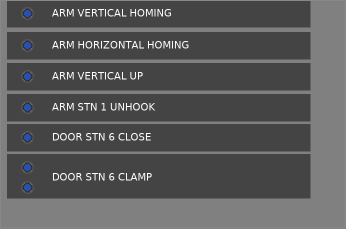
VISUALIZATION Popup_OriginStatus  // 346x229
    Rectangle (0,0 346x229)
    Rectangle (7,0 303x27)
    Label (49,1 258x24), "ARM VERTICAL HOMING"
    Lamp1 (20,6 15x15), variable: ARbArmVertHomeDone[1], style: Lamp-Lamp1-Blue
    Rectangle (7,32 303x27)
    Label (49,33 256x24), "ARM HORIZONTAL HOMING"
    Lamp1 (20,38 15x15), variable: ARbArmHorzHomeDone[1], style: Lamp-Lamp1-Blue
    Rectangle (7,63 303x27)
    Label (49,64 256x24), "ARM VERTICAL UP"
    Lamp1 (20,69 15x15), variable: ARDSArmCtrl[1].AR3sbPositionCfm[2,1,1], style: Lamp-Lamp1-Blue
    Rectangle (7,94 303x27)
    Label (49,95 259x24), "ARM STN 1 UNHOOK"
    Lamp1 (20,100 15x15), variable: ARDSArmCtrl[1].AR3sbPositionCfm[1,1,7], style: Lamp-Lamp1-Blue
    Rectangle (7,124 303x27)
    Label (49,125 258x24), "DOOR STN 6 CLOSE"
    Lamp1 (20,130 15x15), variable: ARbDI[eX12008_Stn06SlidingDoorRs_Close], style: Lamp-Lamp1-Blue
    Rectangle (7,154 303x44)
    Label (49,165 258x24), "DOOR STN 6 CLAMP"
    Lamp1 (20,160 15x15), variable: ARbDI[eX12100_Stn06SlidingDoorRs01_Clamp], style: Lamp-Lamp1-Blue
    Lamp1 (20,180 15x15), variable: ARbDI[eX12102_Stn06SlidingDoorRs02_Clamp], style: Lamp-Lamp1-Blue
END_VISUALIZATION

(* stored: Version 1.1.0.1, ProductVersion 3.1.4024.12
   Visu Popup_OriginStatus: Id {4f4f93ac-8259-41bd-a337-ead4fc6847dc} *)
